TYPE ST_ShiftCalendarV3 :
STRUCT
    SchemaVersion : UINT;
    UtcOffsetMin : DINT;
    Rows : ARRAY[1..PL_Fraktal.MAX_WEEKLY_SHIFTS] OF ST_ShiftRowV3;
END_STRUCT
END_TYPE

(* stored: Version 1.1.0.1, ProductVersion 3.1.4024.12
   DUT ST_ShiftCalendarV3: Id {7f23d9a5-6b0b-4f50-b97f-fd26c5ec1480} *)
